# EPICS alarm handler configuration: mps_database/bare/alarms/areas/mpln_unds_mp06.alhConfig
GROUP NULL MPLN:UNDS:MP06:1
$ALIAS MPS Link Node 214
$GUIDANCE
LTUH MPS
   Group Name: MPLN:UNDS:MP06:1
   Summary PV:  MPLN:UNDS:MP06:1:STATSUMY
$END
CHANNEL  MPLN:UNDS:MP06:1    MPLN:UNDS:MP06:1:MPS_EN_RBV		-----
CHANNEL  MPLN:UNDS:MP06:1    MPLN:UNDS:MP06:1:LC1_MODE_RBV		-----
